FUNCTION_BLOCK SP_Fill (* Fill parameters (Depth [mm] 0.0..50.0, default 50.0): OPC UA IDs, range check and latching *)
  (* Standard: 61499-2 *)
  (* Version 0.1, 2026-09-28, Project contributors, AAU Smart Production Lab *)
  PACKAGE filler;
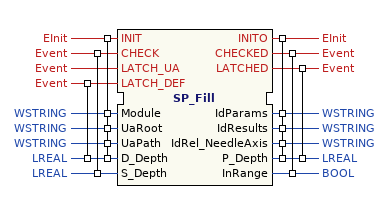
  EVENT_INPUT
    INIT : EInit WITH Module, UaRoot, UaPath, D_Depth;
    CHECK WITH S_Depth;
    LATCH_UA;
    LATCH_DEF WITH D_Depth;
  END_EVENT
  EVENT_OUTPUT
    INITO : EInit WITH IdParams, IdResults, IdRel_NeedleAxis, P_Depth;
    CHECKED WITH InRange;
    LATCHED WITH P_Depth;
  END_EVENT
  VAR_INPUT
    Module : WSTRING;
    UaRoot : WSTRING;
    UaPath : WSTRING;
    D_Depth : LREAL;
    S_Depth : LREAL;
  END_VAR
  VAR_OUTPUT
    IdParams : WSTRING;
    IdResults : WSTRING;
    IdRel_NeedleAxis : WSTRING;
    P_Depth : LREAL;
    InRange : BOOL;
  END_VAR
  EC_STATES
    INIT : INIT -> INITO;
    CHECK : CHECK -> CHECKED;
    LATCH_UA : LATCH_UA -> LATCHED;
    LATCH_DEF : LATCH_DEF -> LATCHED;
  END_STATES
  ALGORITHM INIT IN ST:
IdParams := CONCAT(CONCAT(CONCAT("opc_ua[WRITE;", CONCAT(UaRoot, UaPath)), "/Parameters/Depth"), "]");
IdResults := "";
IdRel_NeedleAxis := CONCAT(CONCAT("loc[", Module), "/NeedleAxis/cmd]");
P_Depth := D_Depth;
  END_ALGORITHM
  ALGORITHM CHECK IN ST:
InRange := (S_Depth >= 0.0) AND (S_Depth <= 50.0);
  END_ALGORITHM
  ALGORITHM LATCH_UA IN ST:
P_Depth := S_Depth;
  END_ALGORITHM
  ALGORITHM LATCH_DEF IN ST:
P_Depth := D_Depth;
  END_ALGORITHM
END_FUNCTION_BLOCK
